INTERFACE I_MessageData

PROPERTY DirRoot : POINTER to string(255)
SET
END_SET
END_PROPERTY

PROPERTY ErrorIndex : reference to uint
SET
END_SET
END_PROPERTY

PROPERTY FileRoot : pointer to string(255)
SET
END_SET
END_PROPERTY

PROPERTY LocalTime : pointer to DT
SET
END_SET
END_PROPERTY

PROPERTY MessageIndex : reference to uint
SET
END_SET
END_PROPERTY

PROPERTY MsgList : pointer to ARRAY[1..GVL_MSG_AXIS.MAX_MESSAGE] OF st_message
SET
END_SET
END_PROPERTY

END_INTERFACE

(* stored: Version 1.1.0.1, ProductVersion 3.1.4026.18
   Itf I_MessageData: Id {6b208c40-7ed9-4bd8-b2d1-b409e5eb6c5a}
   Property DirRoot: Id {738fdab4-694e-4384-b44d-cdaba5d2601f}
   Set Set: Id {0ef69ce3-b3d4-4b76-a62f-d804a8f7ea4a}
   Property ErrorIndex: Id {5aab3c7f-4da1-4393-99eb-080b62f5c438}
   Set Set: Id {6e28abea-72d8-4b60-9c98-61bf0f63a0b3}
   Property FileRoot: Id {786aab6b-7b9b-4033-b43f-2353bab04052}
   Set Set: Id {274c3777-c3de-470e-84da-6d3aebbef2e0}
   Property LocalTime: Id {babe0ec3-5aef-43de-8aee-f2d51ce717da}
   Set Set: Id {43410ce0-3414-4b33-af72-222071e6d131}
   Property MessageIndex: Id {322cd776-8b2a-417e-abcf-14f576170799}
   Set Set: Id {59082d8a-7cf6-4f98-84aa-c79b09e8aa8b}
   Property MsgList: Id {07de972d-30a0-46a8-94d7-7a428dbf7326}
   Set Set: Id {c4a59782-7f1d-4bc9-a099-dd4e21d6e4d6} *)
